{attribute 'qualified_only'}
VAR_GLOBAL
END_VAR

(* stored: Version 1.1.0.1, ProductVersion 3.1.4024.16
   GVL Global: Id {0d3c06d0-68ee-4b36-98cb-d60990801dce} *)
